DATA_BLOCK "CheckPositioningOrder_IDB"
VAR
  Index : Int;
END_VAR
BEGIN
END_DATA_BLOCK
